{attribute 'qualified_only'}
{attribute 'strict'}
TYPE ComStateMachine :
(
	Reset := 0,
	Idle := 1,
	Disabled := 2,
	Warning := 3,
	Start := 5,
	Busy := 6,
	Stop := 7,
	Error := 8
) UDINT := Error;
END_TYPE

(* stored: Version 1.1.0.1, ProductVersion 3.1.4022.17
   DUT CommStateMachine: Id {b16d4de3-76c2-4909-95a2-bbb30c741888} *)
